	        70: // Position vertical Axis
	            "gtyp_SSC".Vertical_Axis.di_Target_Position := "gtyp_SSC".di_Pos_Park_Vertical;
	            "gtyp_SSC".Vertical_Axis.x_Start_Positioning := TRUE;

	            IF ("gtyp_SSC".Vertical_Axis.di_Actual_Position <= ("gtyp_SSC".di_Pos_Park_Vertical + "gtyp_SSC".Vertical_Axis.Config.di_Pos_Window))
	                AND ("gtyp_SSC".Vertical_Axis.di_Actual_Position >= ("gtyp_SSC".di_Pos_Park_Vertical - "gtyp_SSC".Vertical_Axis.Config.di_Pos_Window))
	                AND "gtyp_SSC".Vertical_Axis.x_Position_Reached THEN
	                "gtyp_SSC".Vertical_Axis.x_Start_Positioning := FALSE;
	                #li_StepCase := 80;
	            END_IF;

	        80: // Deciding which doing
	            "gtyp_SSC".x_Park_Position_Reached := TRUE;


	            // Statement section ELSE
	        ELSE
	            ;
	    END_CASE;

	ELSE
	    #lx_Init := TRUE;
	END_IF;
END_FUNCTION_BLOCK

FUNCTION_BLOCK "PRG_SLD_Set_Counter_Values"
TITLE = Program Set counter Values SLD
{ S7_Optimized_Access := 'TRUE' }
AUTHOR : 'A.Schaefer'
VERSION : 0.0
   VAR
      lx_Init { ExternalAccessible := 'False'; ExternalVisible := 'False'; ExternalWritable := 'False'} : Bool;
      lfb_R_Trig_Calib_activ {InstructionName := 'R_TRIG'; LibVersion := '1.0'; ExternalAccessible := 'False'; ExternalVisible := 'False'; ExternalWritable := 'False'; S7_SetPoint := 'False'} : R_TRIG;
   END_VAR


BEGIN
	IF #lx_Init THEN

	    // Reload act. Counter Values
	    IF NOT "gtyp_Setup".x_Counter_Value_Calibration THEN
	        "gtyp_Setup".i_Calib_CounterValue_Blue := "gtyp_SLD".i_CounterValue_Blue;
	        "gtyp_Setup".i_Calib_CounterValue_Red := "gtyp_SLD".i_CounterValue_Red;
	        "gtyp_Setup".i_Calib_CounterValue_White := "gtyp_SLD".i_CounterValue_White;
	    END_IF;

	    // Set Counter Values
	    IF "gtyp_Setup".x_Set_CounterValues AND "gtyp_Setup".x_Counter_Value_Calibration THEN
	        "gtyp_SLD".i_CounterValue_Blue := "gtyp_Setup".i_Calib_CounterValue_Blue;
	        "gtyp_SLD".i_CounterValue_Red := "gtyp_Setup".i_Calib_CounterValue_Red;
	        "gtyp_SLD".i_CounterValue_White := "gtyp_Setup".i_Calib_CounterValue_White;
	        "gtyp_Setup".x_Set_CounterValues := FALSE;
	    END_IF;

	ELSE
	    #lx_Init := TRUE;
	END_IF;
END_FUNCTION_BLOCK

FUNCTION_BLOCK "PRG_VGR_Set_Park_Position"
TITLE = Program Set Positioning VGR
{ S7_Optimized_Access := 'TRUE' }
AUTHOR : 'A.Schaefer'
VERSION : 0.0
   VAR
      lx_Init { ExternalAccessible := 'False'; ExternalVisible := 'False'; ExternalWritable := 'False'} : Bool;
      lx_Start_TON_Wait { ExternalAccessible := 'False'; ExternalVisible := 'False'; ExternalWritable := 'False'} : Bool;
      lt_TON_Wait { ExternalAccessible := 'False'; ExternalVisible := 'False'; ExternalWritable := 'False'} : Time;
      li_StepCase { ExternalAccessible := 'False'; ExternalVisible := 'False'; ExternalWritable := 'False'} : Int;
      lfb_TON_Wait {InstructionName := 'TON_TIME'; LibVersion := '1.0'; ExternalAccessible := 'False'; ExternalVisible := 'False'; ExternalWritable := 'False'; S7_SetPoint := 'False'} : TON_TIME;
      lfb_R_Trig_Start_Park_Pos {InstructionName := 'R_TRIG'; LibVersion := '1.0'; ExternalAccessible := 'False'; ExternalVisible := 'False'; ExternalWritable := 'False'; S7_SetPoint := 'False'} : R_TRIG;
   END_VAR


BEGIN
	IF #lx_Init THEN

	    // FB TON Wait
	    #lfb_TON_Wait(IN := #lx_Start_TON_Wait,
	                  PT := #lt_TON_Wait);

	    #lfb_R_Trig_Start_Park_Pos(CLK := "gtyp_Setup".x_Park_Position
	                               OR "IX_Set_Park_Position");

	    // Set Start Park Position
	    IF #lfb_R_Trig_Start_Park_Pos.Q THEN
	        "gtyp_VGR".x_Start_Park_Position := TRUE;
	        #li_StepCase := 0;
	    END_IF;

	    // not Start Park Pos Step 0
	    IF NOT "gtyp_VGR".x_Start_Park_Position THEN
	        #li_StepCase := 0;
	    END_IF;

	    // step chain HBW
	    CASE #li_StepCase OF

	        0:  // init
	            #lx_Start_TON_Wait := FALSE;
	            #li_StepCase := 10;

	        10:  // Set Positioning activ?
	            IF "gtyp_VGR".x_Start_Park_Position AND NOT "gtyp_VGR".x_Park_Position_Reached THEN
	                "gtyp_VGR".horizontal_Axis.x_Start_Positioning := FALSE;
	                "gtyp_VGR".vertical_Axis.x_Start_Positioning := FALSE;
	                "gtyp_VGR".rotate_Axis.x_Start_Positioning := FALSE;
	                "gtyp_VGR".horizontal_Axis.x_Reference := FALSE;
	                "gtyp_VGR".vertical_Axis.x_Reference := FALSE;
	                "gtyp_VGR".rotate_Axis.x_Reference := FALSE;
	                "gtyp_VGR".vertical_Axis.i_PWM := 800;
	                #li_StepCase := 20;
	            END_IF;

	        20: // homing vertical axis
	            "gtyp_VGR".vertical_Axis.x_Reference := TRUE;

	            IF NOT "gtyp_VGR".vertical_Axis.x_Referenced THEN
	                #li_StepCase := 30;
	            END_IF;

	        30: // homed vertical axis
	            IF "gtyp_VGR".vertical_Axis.x_Referenced THEN
	                "gtyp_VGR".vertical_Axis.x_Reference := FALSE;
	                #li_StepCase := 40;
	            END_IF;

	        40: // homing horizontal axis
	            "gtyp_VGR".horizontal_Axis.x_Reference := TRUE;

	            IF NOT "gtyp_VGR".horizontal_Axis.x_Referenced THEN
	                #li_StepCase := 50;
	            END_IF;

	        50: // homed horizontal axis
	            IF "gtyp_VGR".horizontal_Axis.x_Referenced THEN
	                "gtyp_VGR".horizontal_Axis.x_Reference := FALSE;
	                #li_StepCase := 60;
	            END_IF;

	        60: // homing rotate axis
	            "gtyp_VGR".rotate_Axis.x_Reference := TRUE;

	            IF NOT "gtyp_VGR".rotate_Axis.x_Referenced THEN
	                #li_StepCase := 70;
	            END_IF;

	        70: // homed rotate axis
	            IF "gtyp_VGR".rotate_Axis.x_Referenced THEN
	                "gtyp_VGR".rotate_Axis.x_Reference := FALSE;
	                #li_StepCase := 80;
	            END_IF;

	        80: // Position rotate Axis
	            "gtyp_VGR".rotate_Axis.di_Target_Position   := "gtyp_VGR".di_Pos_Park_rotate;
	            "gtyp_VGR".rotate_Axis.x_Start_Positioning  := TRUE;

	            IF ("gtyp_VGR".rotate_Axis.di_Actual_Position <= ("gtyp_VGR".di_Pos_Park_rotate + "gtyp_VGR".rotate_Axis.Config.di_Pos_Window))
	                AND ("gtyp_VGR".rotate_Axis.di_Actual_Position >= ("gtyp_VGR".di_Pos_Park_rotate - "gtyp_VGR".rotate_Axis.Config.di_Pos_Window))
	                AND "gtyp_VGR".rotate_Axis.x_Position_Reached THEN
	                "gtyp_VGR".rotate_Axis.x_Start_Positioning := FALSE;
	                #li_StepCase := 90;
	            END_IF;

	        90: // Position horizontal Axis
	            "gtyp_VGR".horizontal_Axis.di_Target_Position := "gtyp_VGR".di_Pos_Park_horizontal;
	            "gtyp_VGR".horizontal_Axis.x_Start_Positioning := TRUE;

	            IF ("gtyp_VGR".horizontal_Axis.di_Actual_Position <= ("gtyp_VGR".di_Pos_Park_horizontal + "gtyp_VGR".horizontal_Axis.Config.di_Pos_Window))
	                AND ("gtyp_VGR".horizontal_Axis.di_Actual_Position >= ("gtyp_VGR".di_Pos_Park_horizontal - "gtyp_VGR".horizontal_Axis.Config.di_Pos_Window))
	                AND "gtyp_VGR".horizontal_Axis.x_Position_Reached THEN
	                "gtyp_VGR".horizontal_Axis.x_Start_Positioning := FALSE;
	                #li_StepCase := 100;
	            END_IF;

	        100: // Position vertical Axis
	            "gtyp_VGR".vertical_Axis.i_PWM := 500;
	            "gtyp_VGR".vertical_Axis.di_Target_Position := "gtyp_VGR".di_Pos_Park_vertical;
	            "gtyp_VGR".vertical_Axis.x_Start_Positioning := TRUE;

	            IF ("gtyp_VGR".vertical_Axis.di_Actual_Position <= ("gtyp_VGR".di_Pos_Park_vertical + "gtyp_VGR".vertical_Axis.Config.di_Pos_Window))
	                AND ("gtyp_VGR".vertical_Axis.di_Actual_Position >= ("gtyp_VGR".di_Pos_Park_vertical - "gtyp_VGR".vertical_Axis.Config.di_Pos_Window))
	                AND "gtyp_VGR".vertical_Axis.x_Position_Reached THEN
	                "gtyp_VGR".vertical_Axis.x_Start_Positioning := FALSE;
	                #li_StepCase := 110;
	            END_IF;

	        110: // Deciding which doing
	            "gtyp_VGR".x_Park_Position_Reached := TRUE;


	            // Statement section ELSE
	        ELSE
	            ;
	    END_CASE;

	ELSE
	    #lx_Init := TRUE;
	END_IF;
END_FUNCTION_BLOCK

FUNCTION_BLOCK "PRG_SSC_Axis_Horizontal"
TITLE = Program Axis horizontal SSC
{ S7_Optimized_Access := 'TRUE' }
AUTHOR : 'A.Schaefer'
VERSION : 0.0
   VAR
      lx_Init { ExternalAccessible := 'False'; ExternalVisible := 'False'; ExternalWritable := 'False'} : Bool;
      lfb_Horizontal_Axis { ExternalAccessible := 'False'; ExternalVisible := 'False'; ExternalWritable := 'False'; S7_SetPoint := 'False'} : "FB_Axis";
   END_VAR


BEGIN
	IF #lx_Init THEN

	    // FB Axis horizontal
	    #lfb_Horizontal_Axis(   ini_Axis                := 4,
	                            indi_Increment          := "gtyp_SSC".Horizontal_Axis.di_Increment,
	                            inx_Ref_Switch          := "IX_SSC_RefSwitchHorizontalAxis_I2",
	                            inx_Referencing         := "gtyp_SSC".Horizontal_Axis.x_Reference,
	                            inx_Start_Positioning   := "gtyp_SSC".Horizontal_Axis.x_Start_Positioning,
	                            indi_Target_Position    := "gtyp_SSC".Horizontal_Axis.di_Target_Position,
	                            ini_PWM               := "gtyp_SSC".Horizontal_Axis.i_PWM,
	                            inouttyp_Config         := "gtyp_SSC".Horizontal_Axis.Config,
	                            inouttyp_Setup          := "gtyp_SetupAxis");

	    "QX_SSC_M2_HorizontalAxisCounterclockwise_Q4"      := #lfb_Horizontal_Axis.outx_Motor_Neg;
	    "QX_SSC_M2_HorizontalAxisClockwise_Q3"             := #lfb_Horizontal_Axis.outx_Motor_Pos;
	    "QW_SSC_PWM_Horizontal_M2"                         := #lfb_Horizontal_Axis.outi_Motor_PWM;
	    "gtyp_SSC".Horizontal_Axis.di_Actual_Position   := #lfb_Horizontal_Axis.outdi_Actual_Position;
	    "gtyp_SSC".Horizontal_Axis.x_Referenced         := #lfb_Horizontal_Axis.outx_Referenced;
	    "gtyp_SSC".Horizontal_Axis.x_Position_Reached   := #lfb_Horizontal_Axis.outx_Position_Reached;
	ELSE
	    #lx_Init := TRUE;
	END_IF;
END_FUNCTION_BLOCK

FUNCTION_BLOCK "PRG_HBW_Set_Park_Position"
TITLE = Program Set Positioning HBW
{ S7_Optimized_Access := 'TRUE' }
AUTHOR : 'A.Schaefer'
VERSION : 0.0
   VAR
      lx_Init { ExternalAccessible := 'False'; ExternalVisible := 'False'; ExternalWritable := 'False'} : Bool;
      lx_Start_TON_Wait { ExternalAccessible := 'False'; ExternalVisible := 'False'; ExternalWritable := 'False'} : Bool;
      lt_TON_Wait { ExternalAccessible := 'False'; ExternalVisible := 'False'; ExternalWritable := 'False'} : Time;
      li_StepCase { ExternalAccessible := 'False'; ExternalVisible := 'False'; ExternalWritable := 'False'} : Int;
      lfb_TON_Wait {InstructionName := 'TON_TIME'; LibVersion := '1.0'; ExternalAccessible := 'False'; ExternalVisible := 'False'; ExternalWritable := 'False'; S7_SetPoint := 'False'} : TON_TIME;
      lfb_R_Trig_Start_Park_Pos {InstructionName := 'R_TRIG'; LibVersion := '1.0'; ExternalAccessible := 'False'; ExternalVisible := 'False'; ExternalWritable := 'False'; S7_SetPoint := 'False'} : R_TRIG;
   END_VAR


BEGIN
	IF #lx_Init THEN

	    // FB TON Wait
	    #lfb_TON_Wait(IN := #lx_Start_TON_Wait,
	                  PT := #lt_TON_Wait);

	    #lfb_R_Trig_Start_Park_Pos(CLK := "gtyp_Setup".x_Park_Position
	                               OR "IX_Set_Park_Position");

	    // Set Start Park Position
	    IF #lfb_R_Trig_Start_Park_Pos.Q THEN
	        "gtyp_HBW".x_Start_Park_Position := TRUE;
	        #li_StepCase := 0;
	    END_IF;

	    // not Start Park Pos Step 0
	    IF NOT "gtyp_HBW".x_Start_Park_Position THEN
	        #li_StepCase := 0;
	    END_IF;

	    // step chain HBW
	    CASE #li_StepCase OF

	        0:  // init
	            #lx_Start_TON_Wait := FALSE;
	            #li_StepCase := 10;

	        10:  // Set Positioning activ?
	            IF "IX_HBW_SwitchCantileverFront_I5" OR NOT "IX_HBW_SwitchCantileverBack_I6" THEN
	                "QX_HBW_M4_CantileverBackward_Q8" := TRUE;
	                "QX_HBW_M4_CantileverForward_Q7" := FALSE;
	            ELSIF NOT "IX_HBW_SwitchCantileverFront_I5" AND "IX_HBW_SwitchCantileverBack_I6" THEN
	                "QX_HBW_M4_CantileverBackward_Q8" := FALSE;
	                "QX_HBW_M4_CantileverForward_Q7" := FALSE;
	                #li_StepCase := 20;
	            END_IF;

	        20:  // Set Positioning activ?
	            IF "gtyp_HBW".x_Start_Park_Position AND NOT "gtyp_HBW".x_Park_Position_Reached THEN
	                "gtyp_HBW".Horizontal_Axis.x_Start_Positioning := FALSE;
	                "gtyp_HBW".Vertical_Axis.x_Start_Positioning := FALSE;
	                "gtyp_HBW".Horizontal_Axis.x_Reference := FALSE;
	                "gtyp_HBW".Vertical_Axis.x_Reference := FALSE;
	                "QX_HBW_M4_CantileverBackward_Q8" := FALSE;
	                "QX_HBW_M4_CantileverForward_Q7" := FALSE;
	                #li_StepCase := 30;
	            END_IF;

	        30: // homing vertical axis
	            "gtyp_HBW".Vertical_Axis.x_Reference := TRUE;

	            IF NOT "gtyp_HBW".Vertical_Axis.x_Referenced THEN
	                #li_StepCase := 40;
	            END_IF;

	        40: // homed vertical axis
	            IF "gtyp_HBW".Vertical_Axis.x_Referenced THEN
	                "gtyp_HBW".Vertical_Axis.x_Reference := FALSE;
	                #li_StepCase := 50;
	            END_IF;

	        50: // homing horizontal axis
	            "gtyp_HBW".Horizontal_Axis.x_Reference := TRUE;

	            IF NOT "gtyp_HBW".Horizontal_Axis.x_Referenced THEN
	                #li_StepCase := 60;
	            END_IF;

	        60: // homed horizontal axis
	            IF "gtyp_HBW".Horizontal_Axis.x_Referenced THEN
	                "gtyp_HBW".Horizontal_Axis.x_Reference := FALSE;
	                #li_StepCase := 70;
	            END_IF;

	        70: // Position horizontal Axis
	            "gtyp_HBW".Horizontal_Axis.di_Target_Position := "gtyp_HBW".di_Pos_Park_Horizontal;
	            "gtyp_HBW".Horizontal_Axis.x_Start_Positioning := TRUE;

	            IF ("gtyp_HBW".Horizontal_Axis.di_Actual_Position <= ("gtyp_HBW".di_Pos_Park_Horizontal + "gtyp_HBW".Horizontal_Axis.Config.di_Pos_Window))
	                AND ("gtyp_HBW".Horizontal_Axis.di_Actual_Position >= ("gtyp_HBW".di_Pos_Park_Horizontal - "gtyp_HBW".Horizontal_Axis.Config.di_Pos_Window))
	                AND "gtyp_HBW".Horizontal_Axis.x_Position_Reached THEN
	                "gtyp_HBW".Horizontal_Axis.x_Start_Positioning := FALSE;
	                #li_StepCase := 80;
	            END_IF;

	        80: // Position vertical Axis
	            "gtyp_HBW".Vertical_Axis.di_Target_Position := "gtyp_HBW".di_Pos_Park_Vertical;
	            "gtyp_HBW".Vertical_Axis.x_Start_Positioning := TRUE;

	            IF ("gtyp_HBW".Vertical_Axis.di_Actual_Position <= ("gtyp_HBW".di_Pos_Park_Vertical + "gtyp_HBW".Vertical_Axis.Config.di_Pos_Window))
	                AND ("gtyp_HBW".Vertical_Axis.di_Actual_Position >= ("gtyp_HBW".di_Pos_Park_Vertical - "gtyp_HBW".Vertical_Axis.Config.di_Pos_Window))
	                AND "gtyp_HBW".Vertical_Axis.x_Position_Reached THEN
	                "gtyp_HBW".Vertical_Axis.x_Start_Positioning := FALSE;
	                #li_StepCase := 90;
	            END_IF;

	        90: // Deciding which doing
	            "gtyp_HBW".x_Park_Position_Reached := TRUE;


	            // Statement section ELSE
	        ELSE
	            ;
	    END_CASE;

	ELSE
	    #lx_Init := TRUE;
	END_IF;
END_FUNCTION_BLOCK

FUNCTION_BLOCK "PRG_Acknowledge"
TITLE = Program Acknowledge
{ S7_Optimized_Access := 'TRUE' }
AUTHOR : 'A.Schaefer'
VERSION : 0.0
   VAR
      lx_Init { ExternalAccessible := 'False'; ExternalVisible := 'False'; ExternalWritable := 'False'} : Bool;
      li_StepCase { ExternalAccessible := 'False'; ExternalVisible := 'False'; ExternalWritable := 'False'} : Int;
      lldt_Ack_old { ExternalAccessible := 'False'; ExternalVisible := 'False'; ExternalWritable := 'False'} : LDT;
      lfb_TON_Wait {InstructionName := 'TON_TIME'; LibVersion := '1.0'; ExternalAccessible := 'False'; ExternalVisible := 'False'; ExternalWritable := 'False'; S7_SetPoint := 'False'} : TON_TIME;
      lx_Start_TON_Wait { ExternalAccessible := 'False'; ExternalVisible := 'False'; ExternalWritable := 'False'} : Bool;
   END_VAR


BEGIN
	IF #lx_Init THEN
	    #lfb_TON_Wait(IN:= #lx_Start_TON_Wait,PT:= T#20s);

	    CASE #li_StepCase OF

	        0:  // Init
	            #lx_Start_TON_Wait := FALSE;

	            // check whether acknowledgment has been pressed (time stamp changes)
	            IF ("gtyp_Interface_Dashboard".Publish.ldt_AcknowledgeButton > #lldt_Ack_old)
	                OR "gtyp_Setup".x_AcknowledgeButton THEN
	                #lldt_Ack_old    := "gtyp_Interface_Dashboard".Publish.ldt_AcknowledgeButton;
	                #li_StepCase    := 10;
	            END_IF;

	        10: // acknowledge Errors
	            "gtyp_HBW".x_Error := FALSE;
	            "gtyp_MPO".x_Error := FALSE;
	            "gtyp_SLD".x_Error := FALSE;
	            #li_StepCase := 20;

	        20: // Reset acknowledge button
	            "gtyp_Setup".x_AcknowledgeButton := FALSE;
	            #li_StepCase := 0;
	    // Statement section ELSE
	    ELSE
	        ;
	    END_CASE;

	ELSE
	    #lx_Init := TRUE;
	END_IF;
END_FUNCTION_BLOCK

FUNCTION_BLOCK "PRG_NFC"
TITLE = Program NFC
{ S7_Optimized_Access := 'TRUE' }
AUTHOR : 'A.Schaefer'
VERSION : 0.0
   VAR
      lx_Init { ExternalAccessible := 'False'; ExternalVisible := 'False'; ExternalWritable := 'False'} : Bool;
      lx_Start { ExternalAccessible := 'False'; ExternalVisible := 'False'; ExternalWritable := 'False'} : Bool;
      lx_Time_Wait { ExternalAccessible := 'False'; ExternalVisible := 'False'; ExternalWritable := 'False'} : Bool;
      lx_Time_Error { ExternalAccessible := 'False'; ExternalVisible := 'False'; ExternalWritable := 'False'} : Bool;
      li_StepCase { ExternalAccessible := 'False'; ExternalVisible := 'False'; ExternalWritable := 'False'} : Int;
      ldt_MQTT { ExternalAccessible := 'False'; ExternalVisible := 'False'; ExternalWritable := 'False'} : Date_And_Time;
      ldt_Delete_old { ExternalAccessible := 'False'; ExternalVisible := 'False'; ExternalWritable := 'False'} : LDT;
      ldt_Read_old { ExternalAccessible := 'False'; ExternalVisible := 'False'; ExternalWritable := 'False'} : LDT;
      li_Return_LDT { ExternalAccessible := 'False'; ExternalVisible := 'False'; ExternalWritable := 'False'} : Int;
      lfb_TON_Error {InstructionName := 'TON_TIME'; LibVersion := '1.0'; ExternalAccessible := 'False'; ExternalVisible := 'False'; ExternalWritable := 'False'; S7_SetPoint := 'False'} : TON_TIME;
      lfb_TON_Wait {InstructionName := 'TON_TIME'; LibVersion := '1.0'; ExternalAccessible := 'False'; ExternalVisible := 'False'; ExternalWritable := 'False'; S7_SetPoint := 'False'} : TON_TIME;
   END_VAR


BEGIN
	IF #lx_Init THEN

	    // runtime monitoring error
	    #lfb_TON_Error(IN:= #lx_Time_Error,
	                   PT:= T#30s);

	    // runtime monitoring read uid
	    #lfb_TON_Wait(IN := #lx_Time_Wait,
	                  PT := T#5s);

	     // step chain NFC
	    CASE #li_StepCase OF

	        0:  // init
	            #lx_Time_Wait                := FALSE;
	            "gtyp_VGR"."x_NFC_Completed" := FALSE;

	            // delete and write first state to chip
	            IF "gtyp_VGR".x_NFC_Start_First AND NOT "gtyp_VGR".x_Workpiece_NiO THEN
	                "gtyp_Interface_TXT_Controler".Subscribe.State_NFC_Device.Workpiece.s_state := '';
	                "gtyp_Interface_TXT_Controler".Subscribe.State_NFC_Device.Workpiece.s_type := '';

	                "gtyp_Interface_TXT_Controler".Publish.ActionButtonNFCModule.s_cmd := '';
	                #li_StepCase := 10;
	                // write color or processed finished to chip
	            ELSIF "gtyp_VGR".x_NFC_Start AND NOT "gtyp_VGR".x_Workpiece_NiO THEN
	                "gtyp_Interface_TXT_Controler".Publish.ActionButtonNFCModule.s_cmd := '';
	                #li_StepCase := 40;
	                // read chip for delete HBW
	            ELSIF "QX_SSC_LED_Green_Q5" AND NOT "gtyp_VGR".x_Workpiece_NiO THEN
	                #ldt_Read_old := "gtyp_Interface_Dashboard".Publish.ActionButtonNFCModule.ldt_ts;
	                "gtyp_VGR".x_NFC_Start_First := FALSE;
	                "gtyp_VGR".x_NFC_Start := FALSE;
	                "gtyp_Interface_TXT_Controler".Publish.ActionButtonNFCModule.s_cmd := '';
	                #li_StepCase := 60;
	            END_IF;

	        10: // delete

	            "gtyp_Interface_TXT_Controler".Publish.ActionButtonNFCModule.s_cmd := 'delete';
	            #li_Return_LDT := RD_SYS_T(#ldt_MQTT);
	            "gtyp_Interface_TXT_Controler".Publish.ActionButtonNFCModule.ldt_ts := DT_TO_LDT(#ldt_MQTT);

	            #li_StepCase := 20;

	        20: // wait to answer from dashboard
	            #lx_Time_Error := TRUE;
	            IF ("gtyp_Interface_TXT_Controler".Subscribe.State_NFC_Device.ldt_ts > "gtyp_Interface_TXT_Controler".Publish.ActionButtonNFCModule.ldt_ts)
	                AND ("gtyp_Interface_TXT_Controler".Subscribe.State_NFC_Device.Workpiece.s_type = 'NONE')
	                AND ("gtyp_Interface_TXT_Controler".Subscribe.State_NFC_Device.Workpiece.s_state <> '')
	                AND ("gtyp_Interface_TXT_Controler".Subscribe.State_NFC_Device.Workpiece.s_id <> '') THEN
	                "gtyp_VGR".Workpiece.s_id := "gtyp_Interface_TXT_Controler".Subscribe.State_NFC_Device.Workpiece.s_id;
	                #lx_Time_Error := FALSE;
	                #li_StepCase := 30;
	            END_IF;
	            // runtime error
	            IF #lfb_TON_Error.Q THEN
	                #lx_Time_Error := FALSE;
	                "gtyp_VGR".x_Workpiece_NiO := TRUE;
	                #li_StepCase := 0;
	            END_IF;


	        30: // wait of answer
	            IF "gtyp_Interface_TXT_Controler".Subscribe.State_NFC_Device.Workpiece.s_id <> '' THEN
	                #li_StepCase := 40;
	            END_IF;

	        40:  // write
	            "gtyp_Interface_TXT_Controler".Publish.ActionButtonNFCModule.History            := "gtyp_VGR".History;
	            "gtyp_Interface_TXT_Controler".Publish.ActionButtonNFCModule.Workpiece.s_type   := "gtyp_VGR".Workpiece.s_type;
	            "gtyp_Interface_TXT_Controler".Publish.ActionButtonNFCModule.Workpiece.s_state  := "gtyp_VGR".Workpiece.s_state;

	            #li_Return_LDT := RD_SYS_T(#ldt_MQTT);

	            "gtyp_Interface_TXT_Controler".Publish.ActionButtonNFCModule.s_cmd  := 'write';
	            "gtyp_Interface_TXT_Controler".Publish.ActionButtonNFCModule.ldt_ts := DT_TO_LDT(#ldt_MQTT);

	            #li_StepCase := 50;

	        50: // wait of answer write
	            #lx_Time_Error := TRUE;
	            IF ("gtyp_Interface_TXT_Controler".Subscribe.State_NFC_Device.ldt_ts > "gtyp_Interface_TXT_Controler".Publish.ActionButtonNFCModule.ldt_ts) THEN
	                #lx_Time_Error := FALSE;
	                #li_StepCase := 80;
	            END_IF;
	            // runtime error
	            IF #lfb_TON_Error.Q THEN
	                #lx_Time_Error := FALSE;
	                "gtyp_VGR".x_Workpiece_NiO := TRUE;
	                #li_StepCase := 0;
	            END_IF;

	        60: // read uid cmd

	            #li_Return_LDT := RD_SYS_T(#ldt_MQTT);

	            "gtyp_Interface_TXT_Controler".Publish.ActionButtonNFCModule.s_cmd := 'read_uid';
	            "gtyp_Interface_TXT_Controler".Publish.ActionButtonNFCModule.ldt_ts := DT_TO_LDT(#ldt_MQTT);
	            #lx_Time_Wait   := TRUE;
	            #li_StepCase    := 70;

	        70: // wait of answer read_uid
	            IF NOT "QX_SSC_LED_Green_Q5" OR #lfb_TON_Wait.Q OR ("gtyp_Interface_TXT_Controler".Subscribe.State_NFC_Device.ldt_ts > "gtyp_Interface_TXT_Controler".Publish.ActionButtonNFCModule.ldt_ts) THEN
	                IF LEN("gtyp_Interface_TXT_Controler".Subscribe.State_NFC_Device.Workpiece.s_id) = 8 THEN
	                    "gtyp_Setup".x_Clean_Rack_HBW := TRUE;
	                END_IF;
	                #lx_Time_Wait := FALSE;
	                "gtyp_Interface_TXT_Controler".Subscribe.State_NFC_Device.Workpiece.s_id := '';
	                #li_StepCase := 0;
	            END_IF;

	        80: // completed

	            "gtyp_VGR"."x_NFC_Completed" := TRUE;

	            IF NOT "gtyp_VGR".x_NFC_Start AND NOT "gtyp_VGR".x_NFC_Start_First THEN
	                "gtyp_VGR"."x_NFC_Completed" := FALSE;
	                #lx_Start := FALSE;
	                #li_StepCase := 0;
	            END_IF;

	            // Statement section ELSE
	            ELSE
	                ;
	    END_CASE;

	ELSE
	    #lx_Init := TRUE;
	END_IF;
END_FUNCTION_BLOCK

DATA_BLOCK "PRG_VGR_Axis_vertical_DB"
{ S7_Optimized_Access := 'TRUE' }
VERSION : 0.1
NON_RETAIN
"PRG_VGR_Axis_vertical"

BEGIN

END_DATA_BLOCK

DATA_BLOCK "PRG_VGR_Ablauf_DB"
{ S7_Optimized_Access := 'TRUE' }
VERSION : 0.1
NON_RETAIN
"PRG_VGR_Ablauf"

BEGIN

END_DATA_BLOCK

DATA_BLOCK "PRG_VGR_Axis_horizontal_DB"
{ S7_Optimized_Access := 'TRUE' }
VERSION : 0.1
NON_RETAIN
"PRG_VGR_Axis_horizontal"

BEGIN

END_DATA_BLOCK

DATA_BLOCK "PRG_SSC_Axis_Vertical_DB"
{ S7_Optimized_Access := 'TRUE' }
VERSION : 0.1
NON_RETAIN
"PRG_SSC_Axis_Vertical"

BEGIN

END_DATA_BLOCK

DATA_BLOCK "PRG_SSC_Light_DB"
{ S7_Optimized_Access := 'TRUE' }
VERSION : 0.1
NON_RETAIN
"PRG_SSC_Light"

BEGIN

END_DATA_BLOCK

DATA_BLOCK "PRG_NFC_DB"
{ S7_Optimized_Access := 'TRUE' }
VERSION : 0.1
NON_RETAIN
"PRG_NFC"

BEGIN

END_DATA_BLOCK

DATA_BLOCK "PRG_SSC_Ablauf_DB"
{ S7_Optimized_Access := 'TRUE' }
VERSION : 0.1
NON_RETAIN
"PRG_SSC_Ablauf"

BEGIN

END_DATA_BLOCK

DATA_BLOCK "PRG_VGR_Axis_rotate_DB"
{ S7_Optimized_Access := 'TRUE' }
VERSION : 0.1
NON_RETAIN
"PRG_VGR_Axis_rotate"

BEGIN

END_DATA_BLOCK

DATA_BLOCK "RT_INFO_scl_OB30"
{ S7_Optimized_Access := 'TRUE' }
VERSION : 0.1
NON_RETAIN
   VAR
      mode { ExternalAccessible := 'False'; ExternalVisible := 'False'; ExternalWritable := 'False'} : UInt;   // Mode 1 = Runtime of a specific OB; 2 = Maximum runtime of a specific OB; 3 = Minimum runtime of a specific OB; 10 = Mean value of the percentage of total runtime used by higher-priority OBs; ...
      obNbr { ExternalAccessible := 'False'; ExternalVisible := 'False'; ExternalWritable := 'False'} : OB_ANY;   // OB to read
      infoData { ExternalAccessible := 'False'; ExternalVisible := 'False'; ExternalWritable := 'False'} : LTime;   // mode 1 --> Runtime in LTIME
      returnValue { ExternalAccessible := 'False'; ExternalVisible := 'False'; ExternalWritable := 'False'} : Int;   // Error information of instruction
   END_VAR


BEGIN
   mode := 1;
   obNbr := 1;

END_DATA_BLOCK

DATA_BLOCK "PRG_SSC_Axis_Horizontal_DB"
{ S7_Optimized_Access := 'TRUE' }
VERSION : 0.1
NON_RETAIN
"PRG_SSC_Axis_Horizontal"

BEGIN

END_DATA_BLOCK

DATA_BLOCK "PRG_SSC_Calibration_Color_DB"
{ S7_Optimized_Access := 'TRUE' }
VERSION : 0.1
NON_RETAIN
"PRG_SSC_Calibration_Color"

BEGIN

END_DATA_BLOCK

DATA_BLOCK "PRG_HBW_Axis_Vertical_DB"
{ S7_Optimized_Access := 'TRUE' }
VERSION : 0.1
NON_RETAIN
"PRG_HBW_Axis_Vertical"

BEGIN

END_DATA_BLOCK

DATA_BLOCK "PRG_SSC_Set_Positioning_DB"
{ S7_Optimized_Access := 'TRUE' }
VERSION : 0.1
NON_RETAIN
"PRG_SSC_Set_Positioning"

BEGIN

END_DATA_BLOCK

DATA_BLOCK "PRG_HBW_Set_Positioning_DB"
{ S7_Optimized_Access := 'TRUE' }
VERSION : 0.1
NON_RETAIN
"PRG_HBW_Set_Positioning"

BEGIN

END_DATA_BLOCK

DATA_BLOCK "PRG_VGR_Set_Positioning_DB"
{ S7_Optimized_Access := 'TRUE' }
VERSION : 0.1
NON_RETAIN
"PRG_VGR_Set_Positioning"

BEGIN

END_DATA_BLOCK

DATA_BLOCK "PRG_SLD_Calibration_Color_DB"
{ S7_Optimized_Access := 'TRUE' }
VERSION : 0.1
NON_RETAIN
"PRG_SLD_Calibration_Color"

BEGIN

END_DATA_BLOCK

DATA_BLOCK "PRG_SLD_Set_Counter_Values_DB"
{ S7_Optimized_Access := 'TRUE' }
VERSION : 0.1
NON_RETAIN
"PRG_SLD_Set_Counter_Values"

BEGIN

END_DATA_BLOCK

DATA_BLOCK "PRG_SSC_Set_Park_Position_DB"
{ S7_Optimized_Access := 'TRUE' }
AUTHOR : 'A.Schaefer'
VERSION : 0.0
NON_RETAIN
"PRG_SSC_Set_Park_Position"

BEGIN

END_DATA_BLOCK

DATA_BLOCK "PRG_VGR_Set_Park_Position_DB"
{ S7_Optimized_Access := 'TRUE' }
AUTHOR : 'A.Schaefer'
VERSION : 0.0
NON_RETAIN
"PRG_VGR_Set_Park_Position"

BEGIN

END_DATA_BLOCK

DATA_BLOCK "PRG_HBW_Set_Park_Position_DB"
{ S7_Optimized_Access := 'TRUE' }
AUTHOR : 'A.Schaefer'
VERSION : 0.0
NON_RETAIN
"PRG_HBW_Set_Park_Position"

BEGIN

END_DATA_BLOCK

DATA_BLOCK "RT_INFO_scl_OB1"
{ S7_Optimized_Access := 'TRUE' }
VERSION : 0.1
NON_RETAIN
   VAR
      mode { ExternalAccessible := 'False'; ExternalVisible := 'False'; ExternalWritable := 'False'} : UInt;   // Mode 1 = Runtime of a specific OB; 2 = Maximum runtime of a specific OB; 3 = Minimum runtime of a specific OB; 10 = Mean value of the percentage of total runtime used by higher-priority OBs; ...
      obNbr { ExternalAccessible := 'False'; ExternalVisible := 'False'; ExternalWritable := 'False'} : OB_ANY;   // OB to read
      infoData { ExternalAccessible := 'False'; ExternalVisible := 'False'; ExternalWritable := 'False'} : LTime;   // mode 1 --> Runtime in LTIME
      returnValue { ExternalAccessible := 'False'; ExternalVisible := 'False'; ExternalWritable := 'False'} : Int;   // Error information of instruction
   END_VAR


BEGIN
   mode := 1;
   obNbr := 1;

END_DATA_BLOCK

DATA_BLOCK "PRG_Acknowledge_DB"
{ S7_Optimized_Access := 'TRUE' }
VERSION : 0.1
NON_RETAIN
"PRG_Acknowledge"

BEGIN

END_DATA_BLOCK

DATA_BLOCK "PRG_DSO_Status_DB"
{ S7_Optimized_Access := 'TRUE' }
VERSION : 0.1
NON_RETAIN
"PRG_DSO_Status"

BEGIN

END_DATA_BLOCK

DATA_BLOCK "PRG_DSI_Status_DB"
{ S7_Optimized_Access := 'TRUE' }
VERSION : 0.1
NON_RETAIN
"PRG_DSI_Status"

BEGIN

END_DATA_BLOCK

DATA_BLOCK "PRG_Order_DB"
{ S7_Optimized_Access := 'TRUE' }
VERSION : 0.1
NON_RETAIN
"PRG_Order"

BEGIN

END_DATA_BLOCK

DATA_BLOCK "PRG_SLD_Ablauf_DB"
{ S7_Optimized_Access := 'TRUE' }
VERSION : 0.1
NON_RETAIN
"PRG_SLD_Ablauf"

BEGIN

END_DATA_BLOCK

DATA_BLOCK "PRG_MPO_Ablauf_DB"
{ S7_Optimized_Access := 'TRUE' }
VERSION : 0.1
NON_RETAIN
"PRG_MPO_Ablauf"

BEGIN

END_DATA_BLOCK

DATA_BLOCK "PRG_MPO_Set_Park_Position_DB"
{ S7_Optimized_Access := 'TRUE' }
AUTHOR : 'A.Schaefer'
VERSION : 0.0
NON_RETAIN
"PRG_MPO_Set_Park_Position"

BEGIN

END_DATA_BLOCK

DATA_BLOCK "PRG_HBW_Axis_Horizontal_DB"
{ S7_Optimized_Access := 'TRUE' }
VERSION : 0.1
NON_RETAIN
"PRG_HBW_Axis_Horizontal"

BEGIN

END_DATA_BLOCK

DATA_BLOCK "PRG_HBW_Ablauf_DB"
{ S7_Optimized_Access := 'TRUE' }
VERSION : 0.1
NON_RETAIN
"PRG_HBW_Ablauf"

BEGIN

END_DATA_BLOCK

ORGANIZATION_BLOCK "Main"
TITLE = "Main Program Sweep (Cycle)"
{ S7_Optimized_Access := 'TRUE' }
AUTHOR : 'A.Schaefer'
VERSION : 0.0

BEGIN
	// current cycle Time OB30
	"RT_INFO_scl_OB30".mode := 1;
	"RT_INFO_scl_OB30".obNbr := 30;
	"RT_INFO_scl_OB30".returnValue := RT_INFO(MODE := "RT_INFO_scl_OB30".mode,
	                                          OB := "RT_INFO_scl_OB30".obNbr,
	                                          INFO := "RT_INFO_scl_OB30".infoData);

	// current cycle Time OB1
	"RT_INFO_scl_OB1".mode := 1;
	"RT_INFO_scl_OB1".obNbr := 1;
	"RT_INFO_scl_OB1".returnValue := RT_INFO(MODE := "RT_INFO_scl_OB1".mode,
	                                         OB := "RT_INFO_scl_OB1".obNbr,
	                                         INFO := "RT_INFO_scl_OB1".infoData);

	// sources SSC
	"PRG_SSC_Ablauf_DB"();
	"PRG_SSC_Set_Positioning_DB"();
	"PRG_SSC_Set_Park_Position_DB"();
	"PRG_SSC_Calibration_Color_DB"();
	"PRG_SSC_Axis_Vertical_DB"();
	"PRG_SSC_Axis_Horizontal_DB"();
	"PRG_SSC_Light_DB"();

	// sources VGR
	"PRG_VGR_Ablauf_DB"();
	"PRG_VGR_Set_Positioning_DB"();
	"PRG_VGR_Set_Park_Position_DB"();
	"PRG_VGR_Axis_horizontal_DB"();
	"PRG_VGR_Axis_vertical_DB"();
	"PRG_VGR_Axis_rotate_DB"();
	"PRG_NFC_DB"();

	// sources HBW
	"PRG_HBW_Ablauf_DB"();
	"PRG_HBW_Set_Positioning_DB"();
	"PRG_HBW_Set_Park_Position_DB"();
	"PRG_HBW_Axis_Vertical_DB"();
	"PRG_HBW_Axis_Horizontal_DB"();

	// sources MPO
	"PRG_MPO_Ablauf_DB"();
	"PRG_MPO_Set_Park_Position_DB"();

	// sources SLD
	"PRG_SLD_Ablauf_DB"();
	"PRG_SLD_Calibration_Color_DB"();
	"PRG_SLD_Set_Counter_Values_DB"();

	// sources input/output
	"PRG_DSI_Status_DB"();
	"PRG_DSO_Status_DB"();

	// sources dashboard
	"PRG_Order_DB"();
	"PRG_Acknowledge_DB"();

END_ORGANIZATION_BLOCK

